(* PLC project Tc2_Utilities.FB_GetOemOfLicenseId Demo, tc3-libraries-kb TwinCAT 3.1 *)
(* stored: creationDateTime 2026-05-10T20:00:00, modificationDateTime 2026-05-10T20:00:00 *)

PROGRAM P_Demo_FB_GetOemOfLicenseId
  VAR
    fbFB_GetOemOfLicenseId : FB_GetOemOfLicenseId;  (* Tc2_Utilities.FB_GetOemOfLicenseId 实例 *)
    arg_bExecute : BOOL;  (* VAR_INPUT bExecute *)
    arg_tTimeout : TIME;  (* VAR_INPUT tTimeout *)
    arg_sNetId : T_AmsNetId;  (* VAR_INPUT sNetId *)
    arg_stLicenseId : GUID;  (* VAR_INPUT stLicenseId *)
    out_bBusy : BOOL;  (* VAR_OUTPUT bBusy *)
    out_bError : BOOL;  (* VAR_OUTPUT bError *)
    out_nErrId : UDINT;  (* VAR_OUTPUT nErrId *)
    out_stOemId : GUID;  (* VAR_OUTPUT stOemId *)
  END_VAR

            // ============================================================
// Tc2_Utilities.FB_GetOemOfLicenseId 演示程序（FB 实例）
// ============================================================
// 验证步骤：
//   1. 引用 Tc2_Utilities（及依赖类型所在库 Tc2_System 等）
//   2. 编译 + 登录
//   3. 按 doc.md 给 arg_* 赋值
//   4. 在线监视 out_* / io_* 输出
// ============================================================

fbFB_GetOemOfLicenseId(
    bExecute := arg_bExecute,
    tTimeout := arg_tTimeout,
    sNetId := arg_sNetId,
    stLicenseId := arg_stLicenseId,
    bBusy => out_bBusy,
    bError => out_bError,
    nErrId => out_nErrId,
    stOemId => out_stOemId
);

          
END_PROGRAM
